FUNCTION_BLOCK E_LOAD (* Event-driven Workpiece Load Selection *)
  (* Standard: 61499-1; Function: GUI; Type: Selection; Description: Color selection *)
  (* Version 0.0, 2004-09-25, JHC, Rockwell Automation, Derived from E_SEL_COLOR. *)
  (* Compiler header: package fb.rt.mva; *)
  (* Compiler Java Sun JDK 1.4.2 *)
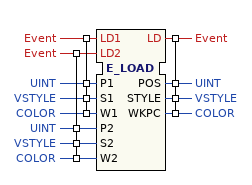
  EVENT_INPUT
    LD1 WITH S1, P1, W1; (* Load Workpiece 1 *)
    LD2 WITH S2, P2, W2; (* Load Workpiece 2 *)
  END_EVENT
  EVENT_OUTPUT
    LD WITH POS, STYLE, WKPC; (* Load Command *)
  END_EVENT
  VAR_INPUT
    P1 : UINT; (* 1 Load Position 1 *)
    S1 : VSTYLE; (* Workpiece 1 Style *)
    W1 : COLOR; (* Workpiece 1 Color *)
    P2 : UINT; (* Load Position 2 *)
    S2 : VSTYLE; (* Workpiece 2 Style *)
    W2 : COLOR; (* Workpiece 2 Color *)
  END_VAR
  VAR_OUTPUT
    POS : UINT; (* Load Position *)
    STYLE : VSTYLE; (* Workpiece Style *)
    WKPC : COLOR; (* Workpiece Color *)
  END_VAR
  ALGORITHM LD1 IN ST: (* Load Workpiece 1 *)
POS := P1;
STYLE := S1;
WKPC := W1;
LD.serviceEvent(this);
  END_ALGORITHM
  ALGORITHM LD2 IN ST: (* Load Workpiece 2 *)
POS := P2;
STYLE := S2;
WKPC := W2;
LD.serviceEvent(this);
  END_ALGORITHM
END_FUNCTION_BLOCK
